// SIMATIC STEP 7 (V5.x) project IoT
// CPU: CPU 315-2 PN/DP
// CPU: CPU 315-2 PN/DP
// station: Hardware
// station: SIMATIC 315(l)
// station: P_ADR_BUS
// station: Hardware
// station: SIMATIC 315(r)
// station: P_ADR_BUS
// program: S7-Programm(1)
// program: S7-Programm(2)

SYMBOL_TABLE
"SEND_DATA"	DB 100	DB 100
"RECV_DATA"	DB 200	DB 200
"TSEND"	FB 63	FB 63	// Send Data
"TRCV"	FB 64	FB 64	// Receive Data
"TCON"	FB 65	FB 65	// Connect
"TDISCON"	FB 66	FB 66	// Disconnect
"TRUE"	M 0.1	BOOL
"Startup"	M 0.3	BOOL
"COMPLETE RESTART"	OB 100	OB 100	// Complete Restart
"TEST_DB"	SFC 24	SFC 24	// Test Data Block
"VAT_1"	VAT 1	
END_SYMBOL_TABLE

FUNCTION_BLOCK FB 1
VERSION : 0.1
VAR_INPUT
  INIT_COM : BOOL ;
  ABORT : BOOL ;
END_VAR
VAR
  CONNECTION_START : BOOL ;
  SR_CONN : BOOL ;
  CON_DONE : BOOL ;
  CON_ERROR : BOOL ;
  CON_BUSY : BOOL ;
  CON_STATUS : WORD ;
  CON_STATUS_SAVE : WORD ;
  SEND_REQ_P : BOOL ;
  SEND_REQ : BOOL ;
  SEND_DONE : BOOL ;
  SEND_BUSY : BOOL ;
  SEND_ERROR : BOOL ;
  SEND_STATUS : WORD ;
  SEND_STATUS_SAVE : WORD ;
  SR_SEND : BOOL ;
  RCV_NDR : BOOL ;
  RCV_BUSY : BOOL ;
  RCV_ERROR : BOOL ;
  RCV_STATUS : WORD ;
  RCV_STATUS_SAVE : WORD ;
  RCV_RLEN_SAVE : INT ;
  RCV_RLEN : INT ;
  SR_ABORT : BOOL ;
  ABORT_P : BOOL ;
  ABORT_BUSY : BOOL ;
  ABORT_DONE : BOOL ;
  ABORT_REQ : BOOL ;
  ABORT_ERROR : BOOL ;
  ABORT_STATUS : WORD ;
  ID : WORD ;
END_VAR
BEGIN
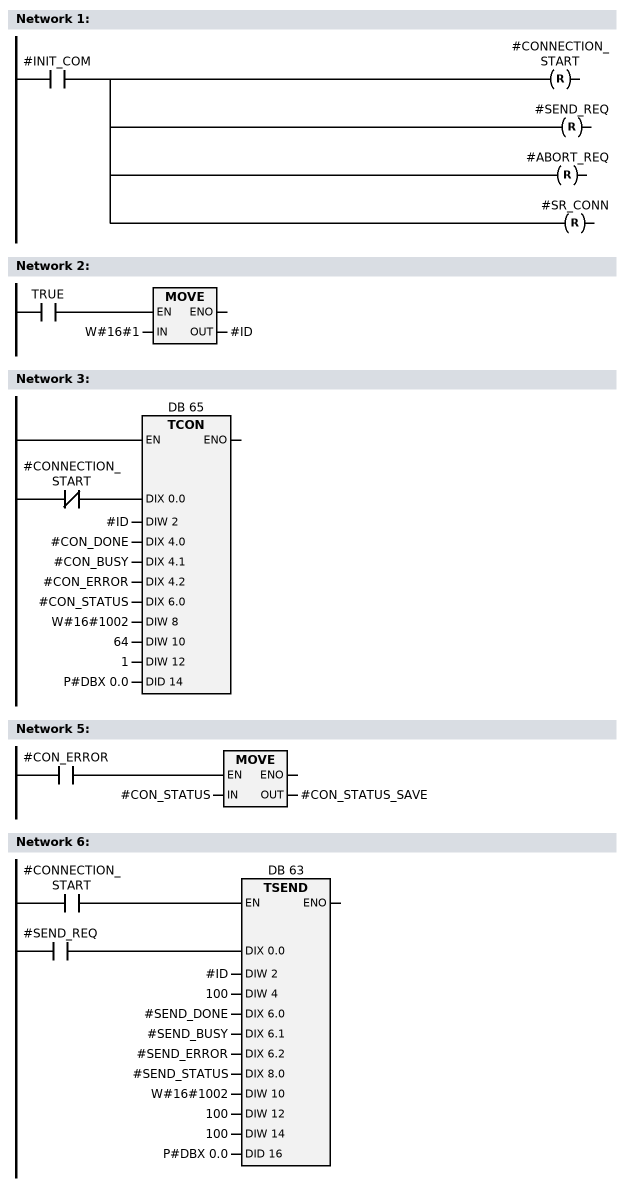
NETWORK
TITLE =
      A     #INIT_COM;
      R     #CONNECTION_START;
      R     #SEND_REQ;
      R     #ABORT_REQ;
      R     #SR_CONN;
NETWORK
TITLE =
      A     "TRUE";
      JNB   _001;
      L     W#16#1;
      T     #ID;
_001: NOP   0;
NETWORK
TITLE =
      AN    #CONNECTION_START;
      =     L 0.0;
      BLD   103;
      CALL  "TCON" , DB 65 (
           DIX 0.0                  := L 0.0,
           DIW 2                    := #ID,
           DIX 4.0                  := #CON_DONE,
           DIX 4.1                  := #CON_BUSY,
           DIX 4.2                  := #CON_ERROR,
           DIX 6.0                  := #CON_STATUS,
           DIW 8                    := W#16#1002,
           DIW 10                   := 64,
           DIW 12                   := 1,
           DID 14                   := P#DBX 0.0);
      NOP   0;
NETWORK
TITLE =
      A(;
      A     #INIT_COM;
      S     #SR_CONN;
      A     #CON_DONE;
      R     #SR_CONN;
      A     #SR_CONN;
      );
      NOT;
      =     #CONNECTION_START;
NETWORK
TITLE =
      A     #CON_ERROR;
      JNB   _002;
      L     #CON_STATUS;
      T     #CON_STATUS_SAVE;
_002: NOP   0;
NETWORK
TITLE =
      A     #SEND_REQ;
      =     L 0.0;
      BLD   103;
      A     #CONNECTION_START;
      JNB   _003;
      CALL  "TSEND" , DB 63 (
           DIX 0.0                  := L 0.0,
           DIW 2                    := #ID,
           DIW 4                    := 100,
           DIX 6.0                  := #SEND_DONE,
           DIX 6.1                  := #SEND_BUSY,
           DIX 6.2                  := #SEND_ERROR,
           DIX 8.0                  := #SEND_STATUS,
           DIW 10                   := W#16#1002,
           DIW 12                   := 100,
           DIW 14                   := 100,
           DID 16                   := P#DBX 0.0);
_003: NOP   0;
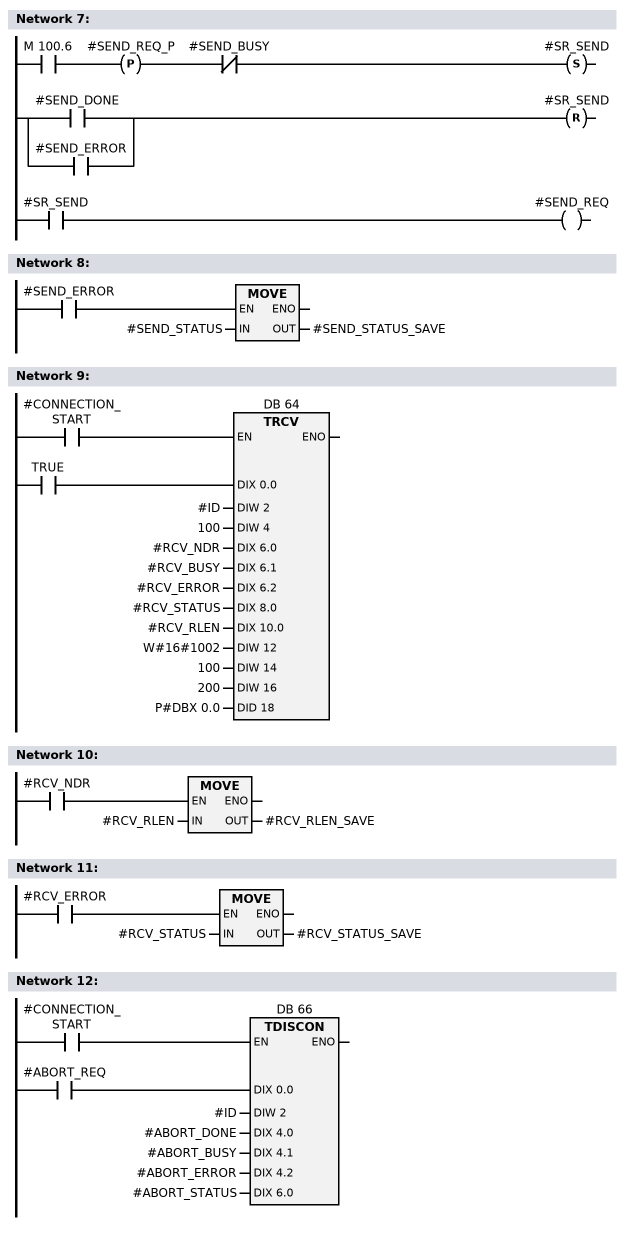
NETWORK
TITLE =
      A     M 100.6;
      FP    #SEND_REQ_P;
      AN    #SEND_BUSY;
      S     #SR_SEND;
      A(;
      O     #SEND_DONE;
      O     #SEND_ERROR;
      );
      R     #SR_SEND;
      A     #SR_SEND;
      =     #SEND_REQ;
NETWORK
TITLE =
      A     #SEND_ERROR;
      JNB   _004;
      L     #SEND_STATUS;
      T     #SEND_STATUS_SAVE;
_004: NOP   0;
NETWORK
TITLE =
      A     "TRUE";
      =     L 0.0;
      BLD   103;
      A     #CONNECTION_START;
      JNB   _005;
      CALL  "TRCV" , DB 64 (
           DIX 0.0                  := L 0.0,
           DIW 2                    := #ID,
           DIW 4                    := 100,
           DIX 6.0                  := #RCV_NDR,
           DIX 6.1                  := #RCV_BUSY,
           DIX 6.2                  := #RCV_ERROR,
           DIX 8.0                  := #RCV_STATUS,
           DIX 10.0                 := #RCV_RLEN,
           DIW 12                   := W#16#1002,
           DIW 14                   := 100,
           DIW 16                   := 200,
           DID 18                   := P#DBX 0.0);
_005: NOP   0;
NETWORK
TITLE =
      A     #RCV_NDR;
      JNB   _006;
      L     #RCV_RLEN;
      T     #RCV_RLEN_SAVE;
_006: NOP   0;
NETWORK
TITLE =
      A     #RCV_ERROR;
      JNB   _007;
      L     #RCV_STATUS;
      T     #RCV_STATUS_SAVE;
_007: NOP   0;
NETWORK
TITLE =
      A     #ABORT_REQ;
      =     L 0.0;
      BLD   103;
      A     #CONNECTION_START;
      JNB   _008;
      CALL  "TDISCON" , DB 66 (
           DIX 0.0                  := L 0.0,
           DIW 2                    := #ID,
           DIX 4.0                  := #ABORT_DONE,
           DIX 4.1                  := #ABORT_BUSY,
           DIX 4.2                  := #ABORT_ERROR,
           DIX 6.0                  := #ABORT_STATUS);
_008: NOP   0;
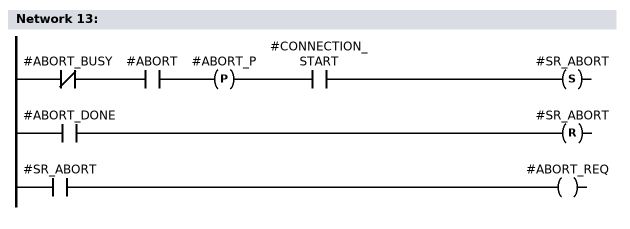
NETWORK
TITLE =
      AN    #ABORT_BUSY;
      A(;
      A     #ABORT;
      FP    #ABORT_P;
      );
      A     #CONNECTION_START;
      S     #SR_ABORT;
      A     #ABORT_DONE;
      R     #SR_ABORT;
      A     #SR_ABORT;
      =     #ABORT_REQ;
END_FUNCTION_BLOCK

// FB 63: know-how protected block, not included

// FB 64: know-how protected block, not included

// FB 65: know-how protected block, not included

// FB 66: know-how protected block, not included

DATA_BLOCK DB 1
TITLE = Connection Parameters for TCON
AUTHOR : SIMATIC
FAMILY : COMM
NAME : TCON_PAR
VERSION : 0.1
  STRUCT
   OUCW_1 : STRUCT
    block_length : WORD  := W#16#40;	//#!Connection_01!#
    id : WORD  := W#16#1;
    connection_type : BYTE  := B#16#12;
    active_est : BOOL  := TRUE;
    local_device_id : BYTE  := B#16#2;
    local_tsap_id_len : BYTE  := B#16#4;
    rem_subnet_id_len : BYTE ;
    rem_staddr_len : BYTE  := B#16#4;
    rem_tsap_id_len : BYTE  := B#16#4;
    next_staddr_len : BYTE ;
    local_tsap_id : ARRAY  [1 .. 16 ] OF BYTE  := B#16#49, B#16#53, B#16#4F, B#16#31, B#16#0, B#16#0, B#16#0, B#16#0, B#16#0, B#16#0, B#16#0, B#16#0, B#16#0, B#16#0, B#16#0, B#16#0;
    rem_subnet_id : ARRAY  [1 .. 6 ] OF BYTE  := B#16#0, B#16#0, B#16#0, B#16#0, B#16#0, B#16#0;
    rem_staddr : ARRAY  [1 .. 6 ] OF BYTE  := B#16#C0, B#16#A8, B#16#0, B#16#1E, B#16#0, B#16#0;
    rem_tsap_id : ARRAY  [1 .. 16 ] OF BYTE  := B#16#49, B#16#53, B#16#4F, B#16#31, B#16#0, B#16#0, B#16#0, B#16#0, B#16#0, B#16#0, B#16#0, B#16#0, B#16#0, B#16#0, B#16#0, B#16#0;
    next_staddr : ARRAY  [1 .. 6 ] OF BYTE  := B#16#0, B#16#0, B#16#0, B#16#0, B#16#0, B#16#0;
    spare : WORD ;	//#!Connection_01!#
   END_STRUCT ;
  END_STRUCT ;	
BEGIN
   OUCW_1.block_length := W#16#40;
   OUCW_1.id := W#16#1;
   OUCW_1.connection_type := B#16#12;
   OUCW_1.active_est := TRUE;
   OUCW_1.local_device_id := B#16#2;
   OUCW_1.local_tsap_id_len := B#16#4;
   OUCW_1.rem_staddr_len := B#16#4;
   OUCW_1.rem_tsap_id_len := B#16#4;
   OUCW_1.local_tsap_id[1] := B#16#49;
   OUCW_1.local_tsap_id[2] := B#16#53;
   OUCW_1.local_tsap_id[3] := B#16#4F;
   OUCW_1.local_tsap_id[4] := B#16#31;
   OUCW_1.rem_staddr[1] := B#16#C0;
   OUCW_1.rem_staddr[2] := B#16#A8;
   OUCW_1.rem_staddr[4] := B#16#1E;
   OUCW_1.rem_tsap_id[1] := B#16#49;
   OUCW_1.rem_tsap_id[2] := B#16#53;
   OUCW_1.rem_tsap_id[3] := B#16#4F;
   OUCW_1.rem_tsap_id[4] := B#16#31;
END_DATA_BLOCK

DATA_BLOCK DB 11
VERSION : 0.0
FB 1
BEGIN
END_DATA_BLOCK

DATA_BLOCK DB 63
AUTHOR : SIMATIC
FAMILY : COMM
VERSION : 0.0
"TSEND"
BEGIN
END_DATA_BLOCK

DATA_BLOCK DB 64
AUTHOR : SIMATIC
FAMILY : COMM
VERSION : 0.0
"TRCV"
BEGIN
END_DATA_BLOCK

DATA_BLOCK DB 65
AUTHOR : SIMATIC
FAMILY : COMM
VERSION : 0.0
"TCON"
BEGIN
END_DATA_BLOCK

DATA_BLOCK DB 66
AUTHOR : SIMATIC
FAMILY : COMM
VERSION : 0.0
"TDISCON"
BEGIN
END_DATA_BLOCK

DATA_BLOCK "SEND_DATA"	// DB 100
VERSION : 0.1
  STRUCT
   SEND_DATA : ARRAY  [0 .. 99 ] OF //vorläufige Platzhaltervariable
   BYTE  := B#16#0;
  END_STRUCT ;	
BEGIN
END_DATA_BLOCK

DATA_BLOCK "RECV_DATA"	// DB 200
VERSION : 0.1
  STRUCT
   RECV_DATA : ARRAY  [0 .. 99 ] OF //vorläufige Platzhaltervariable
   BYTE  := B#16#0;
  END_STRUCT ;	
BEGIN
END_DATA_BLOCK

ORGANIZATION_BLOCK OB 1
TITLE = "Main Program Sweep (Cycle)"
VERSION : 0.1
VAR_TEMP
  OB1_EV_CLASS : BYTE ;	//Bits 0-3 = 1 (Coming event), Bits 4-7 = 1 (Event class 1)
  OB1_SCAN_1 : BYTE ;	//1 (Cold restart scan 1 of OB 1), 3 (Scan 2-n of OB 1)
  OB1_PRIORITY : BYTE ;	//Priority of OB Execution
  OB1_OB_NUMBR : BYTE ;	//1 (Organization block 1, OB1)
  OB1_RESERVED_1 : BYTE ;	//Reserved for system
  OB1_RESERVED_2 : BYTE ;	//Reserved for system
  OB1_PREV_CYCLE : INT ;	//Cycle time of previous OB1 scan (milliseconds)
  OB1_MIN_CYCLE : INT ;	//Minimum cycle time of OB1 (milliseconds)
  OB1_MAX_CYCLE : INT ;	//Maximum cycle time of OB1 (milliseconds)
  OB1_DATE_TIME : DATE_AND_TIME ;	//Date and time OB1 started
END_VAR
BEGIN
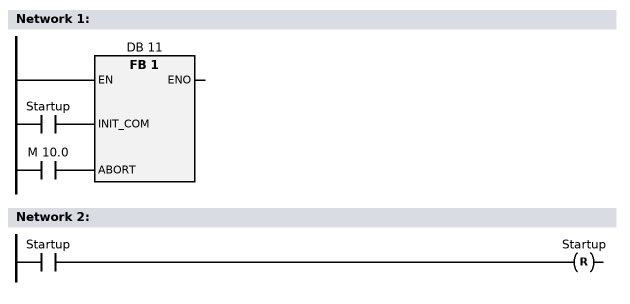
NETWORK
TITLE =
      A     "Startup";
      =     L 20.0;
      BLD   103;
      A     M 10.0;
      =     L 20.1;
      BLD   103;
      CALL  FB 1 , DB 11 (
           INIT_COM                 := L 20.0,
           ABORT                    := L 20.1);
      NOP   0;
NETWORK
TITLE =
      A     "Startup";
      R     "Startup";
NETWORK
TITLE =
END_ORGANIZATION_BLOCK

ORGANIZATION_BLOCK "COMPLETE RESTART"	// OB 100
TITLE = "Complete Restart"
VERSION : 0.1
VAR_TEMP
  OB100_EV_CLASS : BYTE ;	//16#13, Event class 1, Entering event state, Event logged in diagnostic buffer
  OB100_STRTUP : BYTE ;	//16#81/82/83/84 Method of startup
  OB100_PRIORITY : BYTE ;	//Priority of OB Execution
  OB100_OB_NUMBR : BYTE ;	//100 (Organization block 100, OB100)
  OB100_RESERVED_1 : BYTE ;	//Reserved for system
  OB100_RESERVED_2 : BYTE ;	//Reserved for system
  OB100_STOP : WORD ;	//Event that caused CPU to stop (16#4xxx)
  OB100_STRT_INFO : DWORD ;	//Information on how system started
  OB100_DATE_TIME : DATE_AND_TIME ;	//Date and time OB100 started
END_VAR
BEGIN
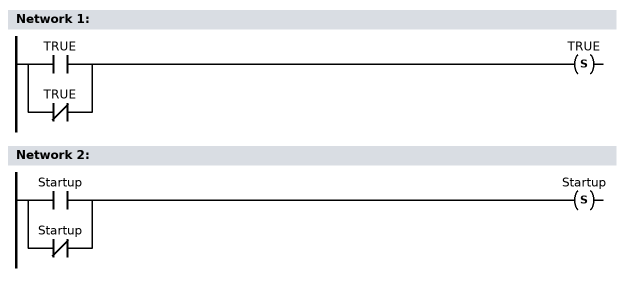
NETWORK
TITLE =
      O     "TRUE";
      ON    "TRUE";
      S     "TRUE";
NETWORK
TITLE =
      O     "Startup";
      ON    "Startup";
      S     "Startup";
END_ORGANIZATION_BLOCK

SYMBOL_TABLE
"SEND_DATA"	DB 100	DB 100
"RECV_DATA"	DB 200	DB 200
"TSEND"	FB 63	FB 63	// Send Data
"TRCV"	FB 64	FB 64	// Receive Data
"TCON"	FB 65	FB 65	// Connect
"TDISCON"	FB 66	FB 66	// Disconnect
"TRUE"	M 0.1	BOOL
"Startup"	M 0.3	BOOL
"COMPLETE RESTART"	OB 100	OB 100	// Complete Restart
"VAT_1"	VAT 1	
END_SYMBOL_TABLE

FUNCTION_BLOCK FB 1
VERSION : 0.1
VAR_INPUT
  INIT_COM : BOOL ;
  ABORT : BOOL ;
END_VAR
VAR
  COMMUNICATION_START : BOOL ;
  CON_DONE : BOOL ;
  CON_BUSY : BOOL ;
  CON_ERROR : BOOL ;
  CON_STATUS : WORD ;
  CON_STATUS_SAVE : WORD ;
  SR_CON : BOOL ;
  SEND_REQ_P : BOOL ;
  SEND_REQ : BOOL ;
  SEND_DONE : BOOL ;
  SEND_BUSY : BOOL ;
  SEND_ERROR : BOOL ;
  SEND_STATUS : WORD ;
  SEND_STATUS_SAVE : WORD ;
  SR_SEND : BOOL ;
  RCV_NDR : BOOL ;
  RCV_BUSY : BOOL ;
  RCV_ERROR : BOOL ;
  RCV_STATUS : WORD ;
  RCV_STATUS_SAVE : WORD ;
  RCV_RLEN : INT ;
  RCV_RLEN_SAVE : INT ;
  ABORT_REQ : BOOL ;
  DIS_DONE : BOOL ;
  DIS_BUSY : BOOL ;
  DIS_ERROR : BOOL ;
  DIS_STATUS : WORD ;
  SR_ABORT : BOOL ;
  ABORT_REQ_P : BOOL ;
  ID : WORD ;
END_VAR
BEGIN
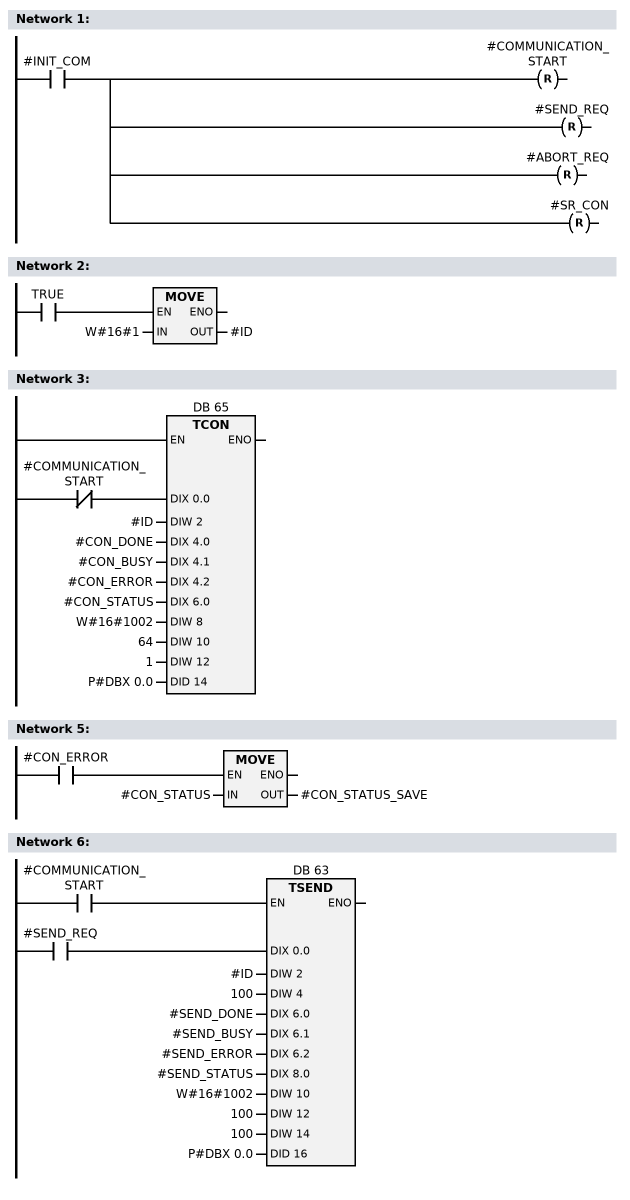
NETWORK
TITLE =
      A     #INIT_COM;
      R     #COMMUNICATION_START;
      R     #SEND_REQ;
      R     #ABORT_REQ;
      R     #SR_CON;
NETWORK
TITLE =
      A     "TRUE";
      JNB   _008;
      L     W#16#1;
      T     #ID;
_008: NOP   0;
NETWORK
TITLE =
      AN    #COMMUNICATION_START;
      =     L 0.0;
      BLD   103;
      CALL  "TCON" , DB 65 (
           DIX 0.0                  := L 0.0,
           DIW 2                    := #ID,
           DIX 4.0                  := #CON_DONE,
           DIX 4.1                  := #CON_BUSY,
           DIX 4.2                  := #CON_ERROR,
           DIX 6.0                  := #CON_STATUS,
           DIW 8                    := W#16#1002,
           DIW 10                   := 64,
           DIW 12                   := 1,
           DID 14                   := P#DBX 0.0);
      NOP   0;
NETWORK
TITLE =
      A(;
      A     #INIT_COM;
      S     #SR_CON;
      A     #CON_DONE;
      R     #SR_CON;
      A     #SR_CON;
      );
      NOT;
      =     #COMMUNICATION_START;
NETWORK
TITLE =
      A     #CON_ERROR;
      JNB   _009;
      L     #CON_STATUS;
      T     #CON_STATUS_SAVE;
_009: NOP   0;
NETWORK
TITLE =
      A     #SEND_REQ;
      =     L 0.0;
      BLD   103;
      A     #COMMUNICATION_START;
      JNB   _00a;
      CALL  "TSEND" , DB 63 (
           DIX 0.0                  := L 0.0,
           DIW 2                    := #ID,
           DIW 4                    := 100,
           DIX 6.0                  := #SEND_DONE,
           DIX 6.1                  := #SEND_BUSY,
           DIX 6.2                  := #SEND_ERROR,
           DIX 8.0                  := #SEND_STATUS,
           DIW 10                   := W#16#1002,
           DIW 12                   := 100,
           DIW 14                   := 100,
           DID 16                   := P#DBX 0.0);
_00a: NOP   0;
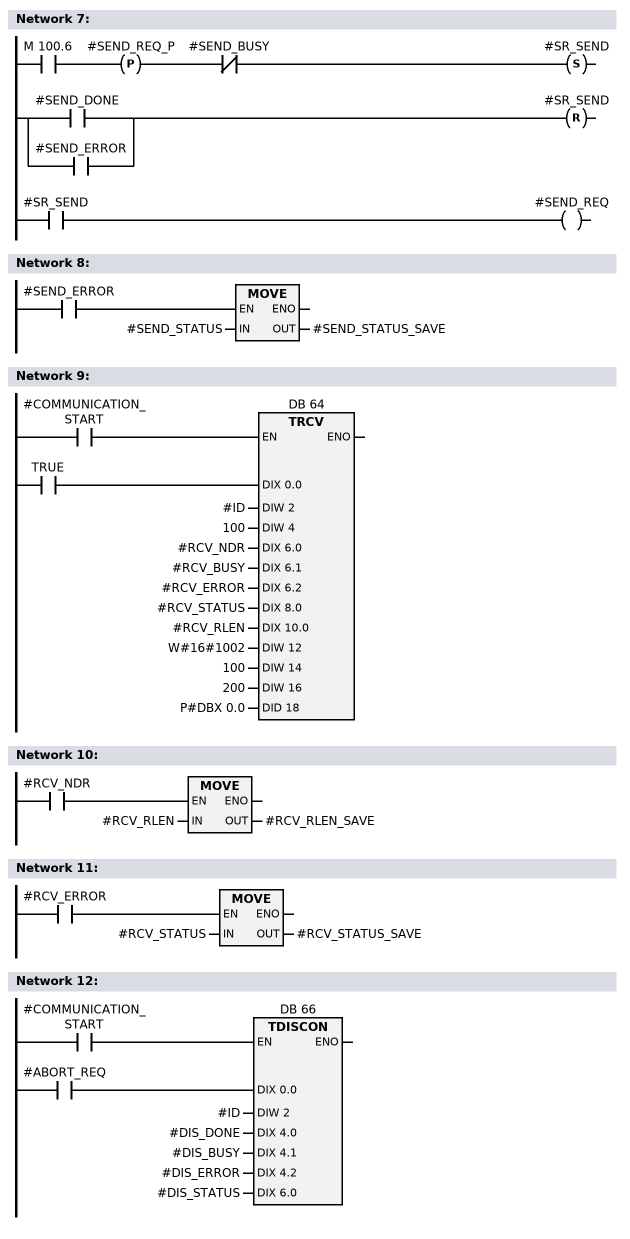
NETWORK
TITLE =
      A     M 100.6;
      FP    #SEND_REQ_P;
      AN    #SEND_BUSY;
      S     #SR_SEND;
      A(;
      O     #SEND_DONE;
      O     #SEND_ERROR;
      );
      R     #SR_SEND;
      A     #SR_SEND;
      =     #SEND_REQ;
NETWORK
TITLE =
      A     #SEND_ERROR;
      JNB   _00b;
      L     #SEND_STATUS;
      T     #SEND_STATUS_SAVE;
_00b: NOP   0;
NETWORK
TITLE =
      A     "TRUE";
      =     L 0.0;
      BLD   103;
      A     #COMMUNICATION_START;
      JNB   _00c;
      CALL  "TRCV" , DB 64 (
           DIX 0.0                  := L 0.0,
           DIW 2                    := #ID,
           DIW 4                    := 100,
           DIX 6.0                  := #RCV_NDR,
           DIX 6.1                  := #RCV_BUSY,
           DIX 6.2                  := #RCV_ERROR,
           DIX 8.0                  := #RCV_STATUS,
           DIX 10.0                 := #RCV_RLEN,
           DIW 12                   := W#16#1002,
           DIW 14                   := 100,
           DIW 16                   := 200,
           DID 18                   := P#DBX 0.0);
_00c: NOP   0;
NETWORK
TITLE =
      A     #RCV_NDR;
      JNB   _00d;
      L     #RCV_RLEN;
      T     #RCV_RLEN_SAVE;
_00d: NOP   0;
NETWORK
TITLE =
      A     #RCV_ERROR;
      JNB   _00e;
      L     #RCV_STATUS;
      T     #RCV_STATUS_SAVE;
_00e: NOP   0;
NETWORK
TITLE =
      A     #ABORT_REQ;
      =     L 0.0;
      BLD   103;
      A     #COMMUNICATION_START;
      JNB   _00f;
      CALL  "TDISCON" , DB 66 (
           DIX 0.0                  := L 0.0,
           DIW 2                    := #ID,
           DIX 4.0                  := #DIS_DONE,
           DIX 4.1                  := #DIS_BUSY,
           DIX 4.2                  := #DIS_ERROR,
           DIX 6.0                  := #DIS_STATUS);
_00f: NOP   0;
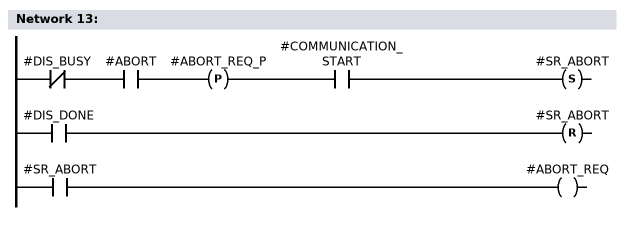
NETWORK
TITLE =
      AN    #DIS_BUSY;
      A(;
      A     #ABORT;
      FP    #ABORT_REQ_P;
      );
      A     #COMMUNICATION_START;
      S     #SR_ABORT;
      A     #DIS_DONE;
      R     #SR_ABORT;
      A     #SR_ABORT;
      =     #ABORT_REQ;
END_FUNCTION_BLOCK

// FB 63: know-how protected block, not included

// FB 64: know-how protected block, not included

// FB 65: know-how protected block, not included

// FB 66: know-how protected block, not included

DATA_BLOCK DB 1
TITLE = Connection Parameters for TCON
AUTHOR : SIMATIC
FAMILY : COMM
NAME : TCON_PAR
VERSION : 0.1
  STRUCT
   OUCW_1 : STRUCT
    block_length : WORD  := W#16#40;	//#!Connection_01!#
    id : WORD  := W#16#1;
    connection_type : BYTE  := B#16#12;
    active_est : BOOL ;
    local_device_id : BYTE  := B#16#2;
    local_tsap_id_len : BYTE  := B#16#4;
    rem_subnet_id_len : BYTE ;
    rem_staddr_len : BYTE  := B#16#4;
    rem_tsap_id_len : BYTE  := B#16#4;
    next_staddr_len : BYTE ;
    local_tsap_id : ARRAY  [1 .. 16 ] OF BYTE  := B#16#49, B#16#53, B#16#4F, B#16#31, B#16#0, B#16#0, B#16#0, B#16#0, B#16#0, B#16#0, B#16#0, B#16#0, B#16#0, B#16#0, B#16#0, B#16#0;
    rem_subnet_id : ARRAY  [1 .. 6 ] OF BYTE  := B#16#0, B#16#0, B#16#0, B#16#0, B#16#0, B#16#0;
    rem_staddr : ARRAY  [1 .. 6 ] OF BYTE  := B#16#C0, B#16#A8, B#16#0, B#16#14, B#16#0, B#16#0;
    rem_tsap_id : ARRAY  [1 .. 16 ] OF BYTE  := B#16#49, B#16#53, B#16#4F, B#16#31, B#16#0, B#16#0, B#16#0, B#16#0, B#16#0, B#16#0, B#16#0, B#16#0, B#16#0, B#16#0, B#16#0, B#16#0;
    next_staddr : ARRAY  [1 .. 6 ] OF BYTE  := B#16#0, B#16#0, B#16#0, B#16#0, B#16#0, B#16#0;
    spare : WORD ;	//#!Connection_01!#
   END_STRUCT ;
  END_STRUCT ;	
BEGIN
   OUCW_1.block_length := W#16#40;
   OUCW_1.id := W#16#1;
   OUCW_1.connection_type := B#16#12;
   OUCW_1.local_device_id := B#16#2;
   OUCW_1.local_tsap_id_len := B#16#4;
   OUCW_1.rem_staddr_len := B#16#4;
   OUCW_1.rem_tsap_id_len := B#16#4;
   OUCW_1.local_tsap_id[1] := B#16#49;
   OUCW_1.local_tsap_id[2] := B#16#53;
   OUCW_1.local_tsap_id[3] := B#16#4F;
   OUCW_1.local_tsap_id[4] := B#16#31;
   OUCW_1.rem_staddr[1] := B#16#C0;
   OUCW_1.rem_staddr[2] := B#16#A8;
   OUCW_1.rem_staddr[4] := B#16#14;
   OUCW_1.rem_tsap_id[1] := B#16#49;
   OUCW_1.rem_tsap_id[2] := B#16#53;
   OUCW_1.rem_tsap_id[3] := B#16#4F;
   OUCW_1.rem_tsap_id[4] := B#16#31;
END_DATA_BLOCK

DATA_BLOCK DB 11
VERSION : 0.0
FB 1
BEGIN
END_DATA_BLOCK

DATA_BLOCK DB 63
AUTHOR : SIMATIC
FAMILY : COMM
VERSION : 0.0
"TSEND"
BEGIN
END_DATA_BLOCK

DATA_BLOCK DB 64
AUTHOR : SIMATIC
FAMILY : COMM
VERSION : 0.0
"TRCV"
BEGIN
END_DATA_BLOCK

DATA_BLOCK DB 65
AUTHOR : SIMATIC
FAMILY : COMM
VERSION : 0.0
"TCON"
BEGIN
END_DATA_BLOCK

DATA_BLOCK DB 66
AUTHOR : SIMATIC
FAMILY : COMM
VERSION : 0.0
"TDISCON"
BEGIN
END_DATA_BLOCK

DATA_BLOCK "SEND_DATA"	// DB 100
VERSION : 0.1
  STRUCT
   SEND_DATA : ARRAY  [0 .. 99 ] OF //vorläufige Platzhaltervariable
   BYTE  := B#16#0;
  END_STRUCT ;	
BEGIN
END_DATA_BLOCK

DATA_BLOCK "RECV_DATA"	// DB 200
VERSION : 0.1
  STRUCT
   RECV_DATA : ARRAY  [0 .. 99 ] OF //vorläufige Platzhaltervariable
   BYTE  := B#16#0;
  END_STRUCT ;	
BEGIN
END_DATA_BLOCK

ORGANIZATION_BLOCK OB 1
TITLE = "Main Program Sweep (Cycle)"
VERSION : 0.1
VAR_TEMP
  OB1_EV_CLASS : BYTE ;	//Bits 0-3 = 1 (Coming event), Bits 4-7 = 1 (Event class 1)
  OB1_SCAN_1 : BYTE ;	//1 (Cold restart scan 1 of OB 1), 3 (Scan 2-n of OB 1)
  OB1_PRIORITY : BYTE ;	//Priority of OB Execution
  OB1_OB_NUMBR : BYTE ;	//1 (Organization block 1, OB1)
  OB1_RESERVED_1 : BYTE ;	//Reserved for system
  OB1_RESERVED_2 : BYTE ;	//Reserved for system
  OB1_PREV_CYCLE : INT ;	//Cycle time of previous OB1 scan (milliseconds)
  OB1_MIN_CYCLE : INT ;	//Minimum cycle time of OB1 (milliseconds)
  OB1_MAX_CYCLE : INT ;	//Maximum cycle time of OB1 (milliseconds)
  OB1_DATE_TIME : DATE_AND_TIME ;	//Date and time OB1 started
END_VAR
BEGIN
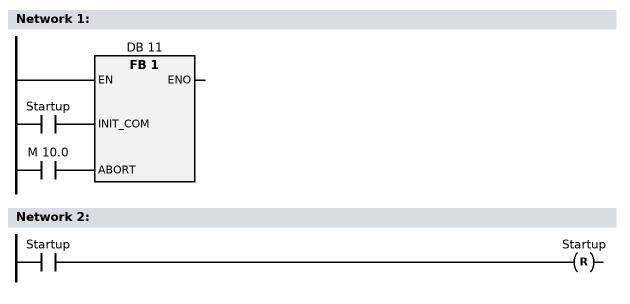
NETWORK
TITLE =
      A     "Startup";
      =     L 20.0;
      BLD   103;
      A     M 10.0;
      =     L 20.1;
      BLD   103;
      CALL  FB 1 , DB 11 (
           INIT_COM                 := L 20.0,
           ABORT                    := L 20.1);
      NOP   0;
NETWORK
TITLE =
      A     "Startup";
      R     "Startup";
END_ORGANIZATION_BLOCK

ORGANIZATION_BLOCK "COMPLETE RESTART"	// OB 100
TITLE = "Complete Restart"
VERSION : 0.1
VAR_TEMP
  OB100_EV_CLASS : BYTE ;	//16#13, Event class 1, Entering event state, Event logged in diagnostic buffer
  OB100_STRTUP : BYTE ;	//16#81/82/83/84 Method of startup
  OB100_PRIORITY : BYTE ;	//Priority of OB Execution
  OB100_OB_NUMBR : BYTE ;	//100 (Organization block 100, OB100)
  OB100_RESERVED_1 : BYTE ;	//Reserved for system
  OB100_RESERVED_2 : BYTE ;	//Reserved for system
  OB100_STOP : WORD ;	//Event that caused CPU to stop (16#4xxx)
  OB100_STRT_INFO : DWORD ;	//Information on how system started
  OB100_DATE_TIME : DATE_AND_TIME ;	//Date and time OB100 started
END_VAR
BEGIN
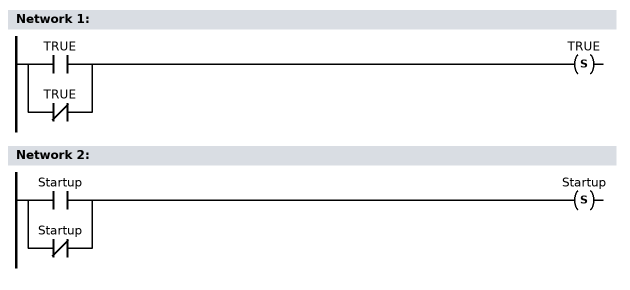
NETWORK
TITLE =
      O     "TRUE";
      ON    "TRUE";
      S     "TRUE";
NETWORK
TITLE =
      O     "Startup";
      ON    "Startup";
      S     "Startup";
END_ORGANIZATION_BLOCK
